TYPE ST_StationPosition :
STRUCT
	fpositionX			: LREAL;
	fpositionY			: LREAL;
END_STRUCT
END_TYPE

(* stored: Version 1.1.0.1, ProductVersion 3.1.4024.12
   DUT ST_StationPosition: Id {9935b2b5-12d7-4bfd-b2bc-e2b928630df8} *)
